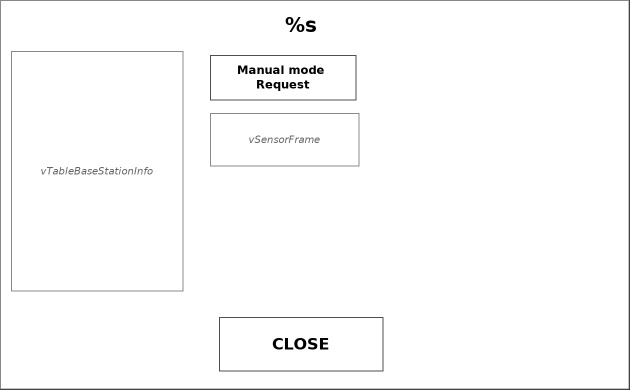
VISUALIZATION vTableLoadingDetail  // 630x390
VAR_IN_OUT
	fbStation:FB_LoadingStation;
	fbTableControl: FB_TableControl;
END_VAR
    Rectangle (0,0 630x390)
    Frame (11,51 172x240)
        shows vTableBaseStationInfo(fbStation := fbStation)
    Rectangle (219,317 164x54), "CLOSE"
        OnMouseDown: execute { fbTableControl.stHMI.iDialogNumber:=0; }
    Rectangle (210,55 146x45), "Manual mode Request", colour toggle: fbStation.bManualModeActive
        toggle fbStation.bManualModeRequest
    Rectangle (226,10 150x30), "%s", text variable: fbStation.sStationName
    Frame (210,113 149x53)
        shows vSensorFrame(iNameIndex := 0, fbSensor := fbStation.fbLoadingSensor)
END_VISUALIZATION

(* stored: Version 1.1.0.1, ProductVersion 3.1.4024.15
   Visu vTableLoadingDetail: Id {dd0cb779-973e-437d-9709-938f12bf3d0f} *)
